Omron Sysmac Studio project distributing_station_with_timer_1.9_attempt (Sysmac Studio 1.54.0.64019, StandardProject)

# Controller new_Controller_0: NJ301-1100 version 1.14
Units and slaves: Node1 : NX-ECC201 (E001); Unit 1 : NX-PC0020 (N1); Unit 2 : NX-ID5442 (N2); Unit 3 : NX-PC0010 (N3); Unit 4 : NX-PC0020 (N4); Unit 5 : NX-OD5121 (N5); Unit 6 : NX-PC0010 (N6); Power Supply : NJ-Px3001; CPU : NJ301-1100; 0 [Unit 0] : CJ1W-AD041-V1 (J01); 1 [Unit 1] : CJ1W-DA041 (J02); 2 : CJ1W-ID211 (J03); 3 : CJ1W-OC211 (J04)
Task PrimaryTask (priority 4, period or condition 1000): Program0

VAR_GLOBAL
    Station_1B2 : BOOL;  (* Ejection Cylinder Extended; at IOBus://rack#0/slot#2/Ch1_In/Ch1_In01; published *)
    Station_1B1 : BOOL;  (* Ejection Cylinder retracted; at IOBus://rack#0/slot#2/Ch1_In/Ch1_In02; published *)
    Station_2B1 : BOOL;  (* Workpiece gripped; at IOBus://rack#0/slot#2/Ch1_In/Ch1_In03; published *)
    Station_3S1 : BOOL;  (* arm_in_magazine; at IOBus://rack#0/slot#2/Ch1_In/Ch1_In04; published *)
    Station_3S2 : BOOL;  (* arm_in_downstream; at IOBus://rack#0/slot#2/Ch1_In/Ch1_In05; published *)
    Station_B4 : BOOL;  (* Magzine empty; at IOBus://rack#0/slot#2/Ch1_In/Ch1_In06; published *)
    Panel_S1 : BOOL;  (* start_button; at IOBus://rack#0/slot#2/Ch1_In/Ch1_In08; published *)
    Panel_S2 : BOOL;  (* stop_button; at IOBus://rack#0/slot#2/Ch1_In/Ch1_In09; published *)
    Panel_S4 : BOOL;  (* reset_button; at IOBus://rack#0/slot#2/Ch1_In/Ch1_In11; published *)
    Station_1Y1 : BOOL;  (* Magzine eject; at IOBus://rack#0/slot#3/Ch1_Out/Ch1_Out00; published *)
    Station_2Y1 : BOOL;  (* Vacuum on; at IOBus://rack#0/slot#3/Ch1_Out/Ch1_Out01; published *)
    Station_2Y2 : BOOL;  (* Ejector_Pulse_On; at IOBus://rack#0/slot#3/Ch1_Out/Ch1_Out02; published *)
    Station_3Y1 : BOOL;  (* arm_2_magazine; at IOBus://rack#0/slot#3/Ch1_Out/Ch1_Out03; published *)
    Station_3Y2 : BOOL;  (* arm_2_downstream; at IOBus://rack#0/slot#3/Ch1_Out/Ch1_Out04; published *)
    Station_H1 : BOOL;  (* start light; at IOBus://rack#0/slot#3/Ch1_Out/Ch1_Out08; published *)
    Station_H2 : BOOL;  (* reset light; at IOBus://rack#0/slot#3/Ch1_Out/Ch1_Out09; published *)
    Panel_H3 : BOOL;  (* Q1 light; at IOBus://rack#0/slot#3/Ch1_Out/Ch1_Out10; published *)
    Panel_H4 : BOOL;  (* Q2 light; at IOBus://rack#0/slot#3/Ch1_Out/Ch1_Out11; published *)
    Station_1B1_in : BOOL;
END_VAR

PROGRAM Program0
VAR
    FB_Panel_1 : FB_Panel;
    run_mode : BOOL;
    stop_mode : BOOL;
    reset_mode : BOOL;
    FB_Actuator_T1_1 : FB_Actuator_T1;
    timer_t1 : TON;
    error_arm : BOOL;
    error_mode : BOOL;
    FB_Actuator_T2_1 : FB_Actuator_T2;
    Piston : RS;
    error_ejec : BOOL;
    extend_piston : BOOL;
    workpiece_ready_set : BOOL;
    flip_flop_1 : RS;
    workpiece_ready : BOOL;
    workpiece_picked_up : BOOL;
    wait_for_piston : TON;
    Workpiece_Checker_1 : Workpiece_Checker;
END_VAR
VAR_EXTERNAL
    Station_3S1 : BOOL;
    Panel_S2 : BOOL;
    Station_3Y2 : BOOL;
    Station_3S2 : BOOL;
    Panel_S1 : BOOL;
    Station_3Y1 : BOOL;
    Panel_S4 : BOOL;
    Station_H1 : BOOL;
    Station_H2 : BOOL;
    Panel_H4 : BOOL;
    Panel_H3 : BOOL;
    Station_1B2 : BOOL;
    Station_1B1 : BOOL;
    Station_1Y1 : BOOL;
    Station_2Y1 : BOOL;
END_VAR
VAR
    _e1 : F_TRIG;
END_VAR

(* Section Section0: ladder, written here as Structured Text *)

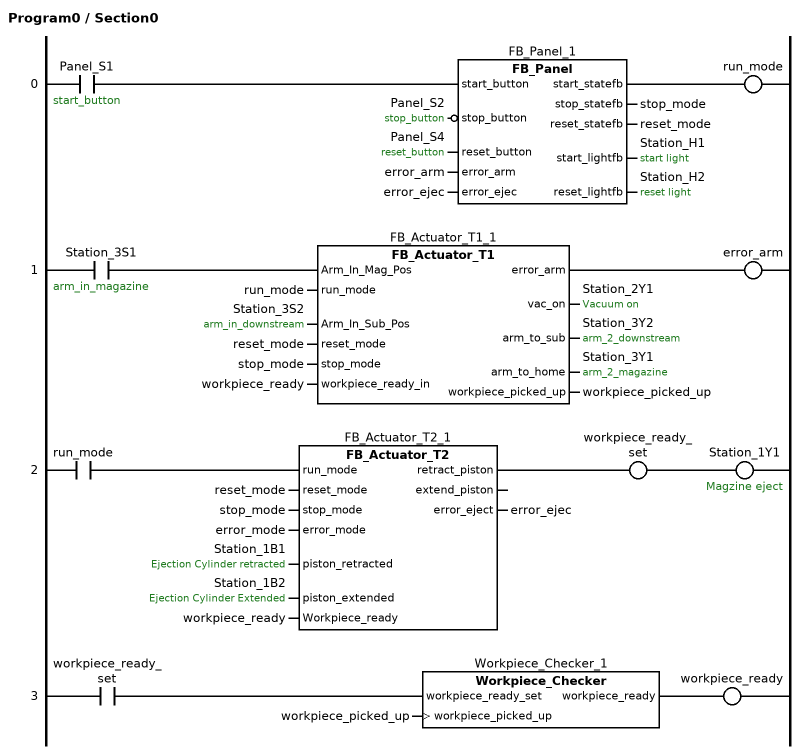
(* Rung 0 *)
FB_Panel_1(start_button := Panel_S1, stop_button := NOT Panel_S2, reset_button := Panel_S4, error_arm := error_arm, error_ejec := error_ejec, stop_statefb => stop_mode, reset_statefb => reset_mode, start_lightfb => Station_H1, reset_lightfb => Station_H2);
run_mode := FB_Panel_1.start_statefb;
(* Rung 1 *)
FB_Actuator_T1_1(Arm_In_Mag_Pos := Station_3S1, run_mode := run_mode, Arm_In_Sub_Pos := Station_3S2, reset_mode := reset_mode, stop_mode := stop_mode, workpiece_ready_in := workpiece_ready, vac_on => Station_2Y1, arm_to_sub => Station_3Y2, arm_to_home => Station_3Y1, workpiece_picked_up => workpiece_picked_up);
error_arm := FB_Actuator_T1_1.error_arm;
(* Rung 2 *)
FB_Actuator_T2_1(run_mode := run_mode, reset_mode := reset_mode, stop_mode := stop_mode, error_mode := error_mode, piston_retracted := Station_1B1, piston_extended := Station_1B2, Workpiece_ready := workpiece_ready, error_eject => error_ejec);
workpiece_ready_set := FB_Actuator_T2_1.retract_piston;
Station_1Y1 := FB_Actuator_T2_1.retract_piston;
(* Rung 3 *)
_e1(CLK := workpiece_picked_up);
Workpiece_Checker_1(workpiece_ready_set := workpiece_ready_set, workpiece_picked_up := _e1.Q);
workpiece_ready := Workpiece_Checker_1.workpiece_ready;
END_PROGRAM

FUNCTION_BLOCK FB_Panel
VAR
    flip_flop : RS;
    flip_flop2 : RS;
    flip_flop_3 : RS;
    flip_flop3 : RS;
    stop_or_error : BOOL;
    error_armfb : BOOL;
    error_q2 : BOOL;
END_VAR
VAR_OUTPUT
    start_statefb : BOOL;
    stop_statefb : BOOL;
    reset_statefb : BOOL;
END_VAR
VAR_INPUT
    start_button : BOOL := False;
    stop_button : BOOL := False;
    reset_button : BOOL := False;
END_VAR
VAR_OUTPUT
    start_lightfb : BOOL;
    reset_lightfb : BOOL;
END_VAR
VAR_INPUT
    error_arm : BOOL;
    error_ejec : BOOL;
END_VAR
VAR_EXTERNAL
    Panel_H4 : BOOL;
END_VAR
(* ladder, written here as Structured Text *)

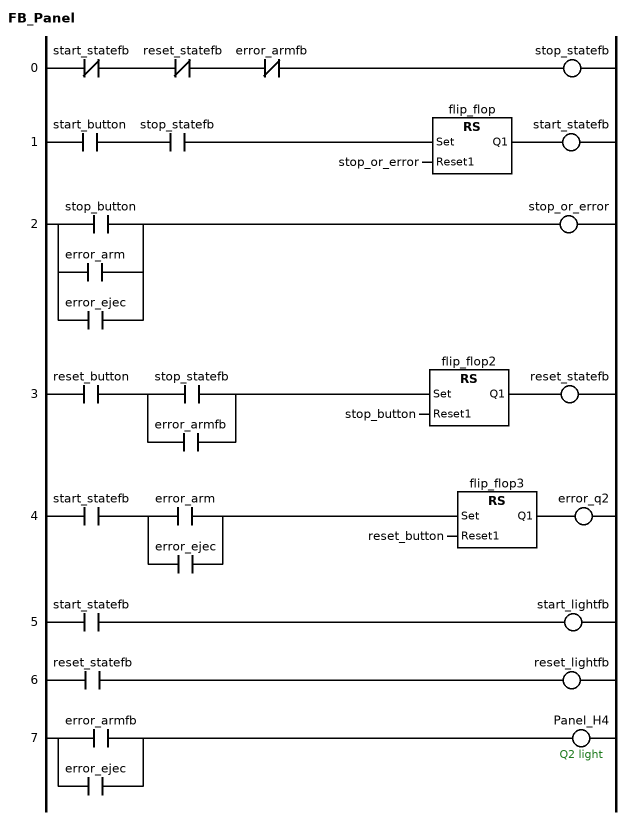
(* Rung 0 *)
stop_statefb := NOT start_statefb AND NOT reset_statefb AND NOT error_armfb;
(* Rung 1 *)
flip_flop(Set := start_button AND stop_statefb, Reset1 := stop_or_error);
start_statefb := flip_flop.Q1;
(* Rung 2 *)
stop_or_error := stop_button OR error_arm OR error_ejec;
(* Rung 3 *)
flip_flop2(Set := reset_button AND (stop_statefb OR error_armfb), Reset1 := stop_button);
reset_statefb := flip_flop2.Q1;
(* Rung 4 *)
flip_flop3(Set := start_statefb AND (error_arm OR error_ejec), Reset1 := reset_button);
error_q2 := flip_flop3.Q1;
(* Rung 5 *)
start_lightfb := start_statefb;
(* Rung 6 *)
reset_lightfb := reset_statefb;
(* Rung 7 *)
Panel_H4 := error_armfb OR error_ejec;
END_FUNCTION_BLOCK

FUNCTION_BLOCK FB_Actuator_T1
VAR
    flip_flop_1 : RS;
    flip_flop_2 : RS;
    reset_to_home : BOOL;
    timer_t1 : TON;
    flip_flop_3 : RS;
    timer_t2 : TON;
    flip_flop_4 : RS;
    error_toSub : BOOL;
    error_toHome : BOOL;
    middle_pos : BOOL;
    middle_timer : AccumulationTimer;
    flip_flop_5 : RS;
    reset_middle : BOOL;
    flip_flop6 : RS;
    move_to_middle_from_home : BOOL;
    move_to_sub : BOOL;
    move_to_home : BOOL;
    move_to_middle_from_sub : BOOL;
    unknown_pos : BOOL;
    reset_vac_arm_to_sub : BOOL;
    timer_t3 : TON;
    t : TIME;
    move_to_su : BOOL;
END_VAR
VAR_INPUT
    Arm_In_Mag_Pos : BOOL;
    run_mode : BOOL;
    Arm_In_Sub_Pos : BOOL;
    reset_mode : BOOL;
    stop_mode : BOOL;
END_VAR
VAR_OUTPUT
    error_arm : BOOL;
END_VAR
VAR_INPUT
    workpiece_ready_in : BOOL;
END_VAR
VAR_OUTPUT
    vac_on : BOOL;
    arm_to_sub : BOOL;
    arm_to_home : BOOL;
    workpiece_picked_up : BOOL;
END_VAR
VAR_EXTERNAL
    Station_3S1 : BOOL;
    Station_3Y1 : BOOL;
    Station_3S2 : BOOL;
    Station_3Y2 : BOOL;
    Station_2Y2 : BOOL;
END_VAR
(* ladder, written here as Structured Text *)

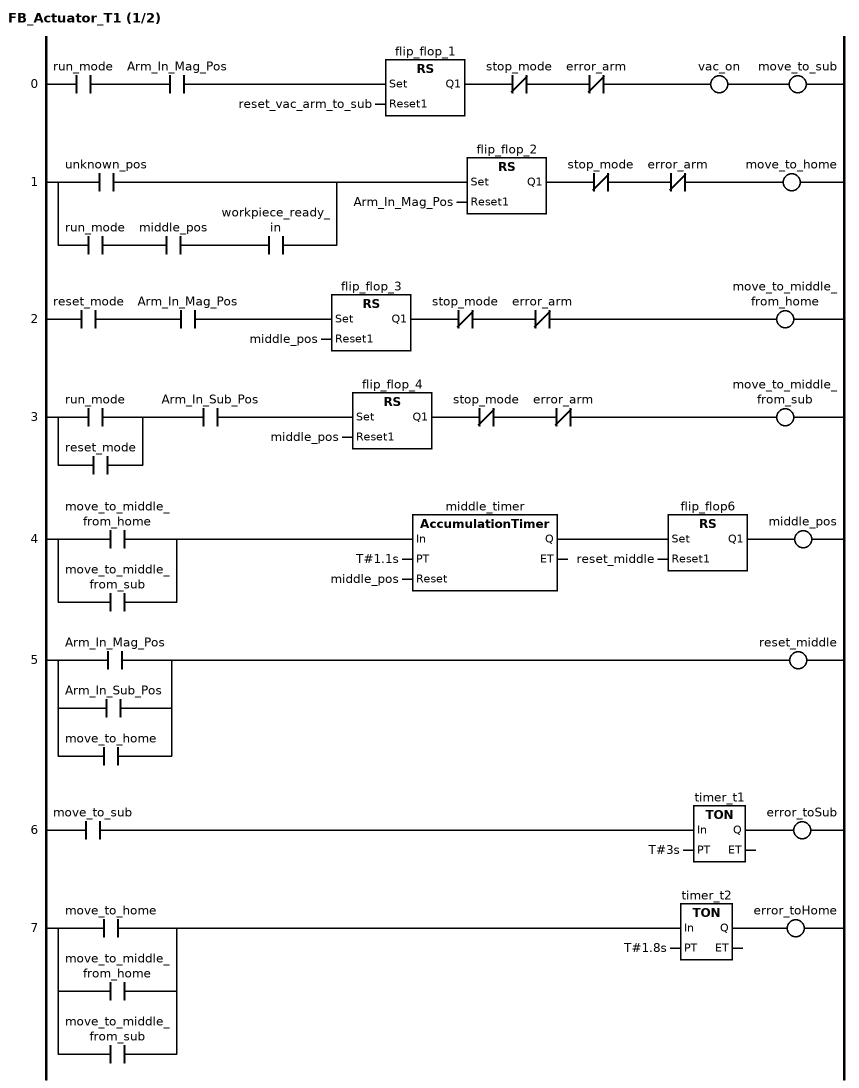
(* Rung 0 *)
flip_flop_1(Set := run_mode AND Arm_In_Mag_Pos, Reset1 := reset_vac_arm_to_sub);
vac_on := flip_flop_1.Q1 AND NOT stop_mode AND NOT error_arm;
move_to_sub := flip_flop_1.Q1 AND NOT stop_mode AND NOT error_arm;
(* Rung 1 *)
flip_flop_2(Set := unknown_pos OR (run_mode AND middle_pos AND workpiece_ready_in), Reset1 := Arm_In_Mag_Pos);
move_to_home := flip_flop_2.Q1 AND NOT stop_mode AND NOT error_arm;
(* Rung 2 *)
flip_flop_3(Set := reset_mode AND Arm_In_Mag_Pos, Reset1 := middle_pos);
move_to_middle_from_home := flip_flop_3.Q1 AND NOT stop_mode AND NOT error_arm;
(* Rung 3 *)
flip_flop_4(Set := (run_mode OR reset_mode) AND Arm_In_Sub_Pos, Reset1 := middle_pos);
move_to_middle_from_sub := flip_flop_4.Q1 AND NOT stop_mode AND NOT error_arm;
(* Rung 4 *)
middle_timer(In := move_to_middle_from_home OR move_to_middle_from_sub, PT := T#1.1s, Reset := middle_pos);
flip_flop6(Set := middle_timer.Q, Reset1 := reset_middle);
middle_pos := flip_flop6.Q1;
(* Rung 5 *)
reset_middle := Arm_In_Mag_Pos OR Arm_In_Sub_Pos OR move_to_home;
(* Rung 6 *)
timer_t1(In := move_to_sub, PT := T#3s);
error_toSub := timer_t1.Q;
(* Rung 7 *)
timer_t2(In := move_to_home OR move_to_middle_from_home OR move_to_middle_from_sub, PT := T#1.8s);
error_toHome := timer_t2.Q;

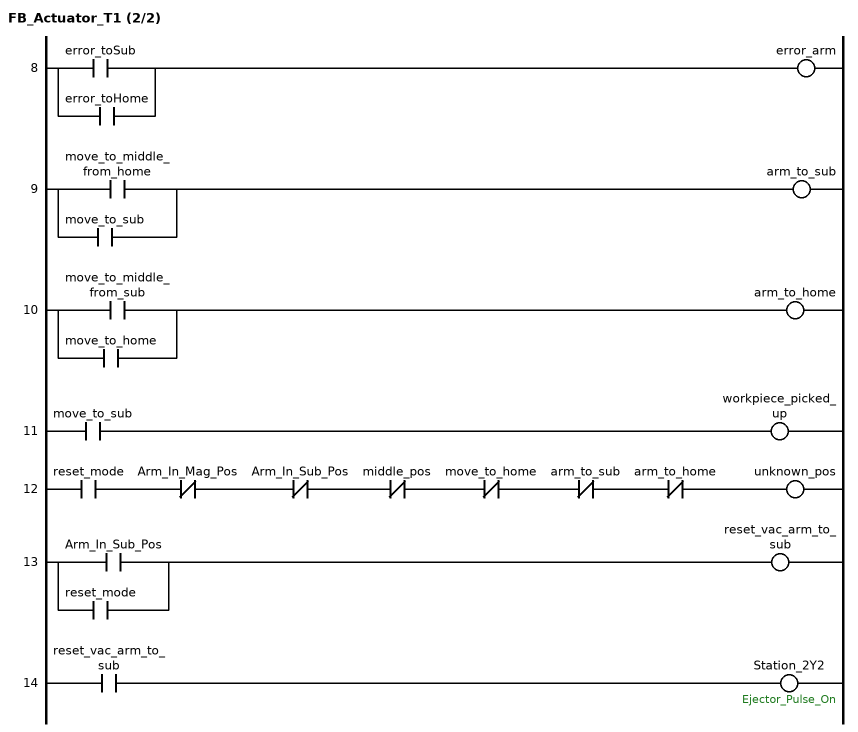
(* Rung 8 *)
error_arm := error_toSub OR error_toHome;
(* Rung 9 *)
arm_to_sub := move_to_middle_from_home OR move_to_sub;
(* Rung 10 *)
arm_to_home := move_to_middle_from_sub OR move_to_home;
(* Rung 11 *)
workpiece_picked_up := move_to_sub;
(* Rung 12 *)
unknown_pos := reset_mode AND NOT Arm_In_Mag_Pos AND NOT Arm_In_Sub_Pos AND NOT middle_pos AND NOT move_to_home AND NOT arm_to_sub AND NOT arm_to_home;
(* Rung 13 *)
reset_vac_arm_to_sub := Arm_In_Sub_Pos OR reset_mode;
(* Rung 14 *)
Station_2Y2 := reset_vac_arm_to_sub;
END_FUNCTION_BLOCK

FUNCTION_BLOCK FB_Actuator_T2
VAR
    reset_to_home : BOOL;
    retract_ff : RS;
    extend_ff : RS;
    extend_t : TON;
    retract_t : TON;
    retract_err : BOOL;
    extend_err : BOOL;
    workpiece_lifted : BOOL;
    Workpiece_ejection : RS;
END_VAR
VAR_INPUT
    run_mode : BOOL;
    reset_mode : BOOL;
    stop_mode : BOOL;
    error_mode : BOOL;
END_VAR
VAR_OUTPUT
    retract_piston : BOOL;
    extend_piston : BOOL;
END_VAR
VAR_INPUT
    piston_retracted : BOOL;
    piston_extended : BOOL;
END_VAR
VAR_OUTPUT
    error_eject : BOOL;
END_VAR
VAR_INPUT
    Workpiece_ready : BOOL;
END_VAR
VAR_EXTERNAL
    Station_B4 : BOOL;
    Station_1B1 : BOOL;
    Station_1B2 : BOOL;
    Station_2Y1 : BOOL;
END_VAR
(* ladder, written here as Structured Text *)

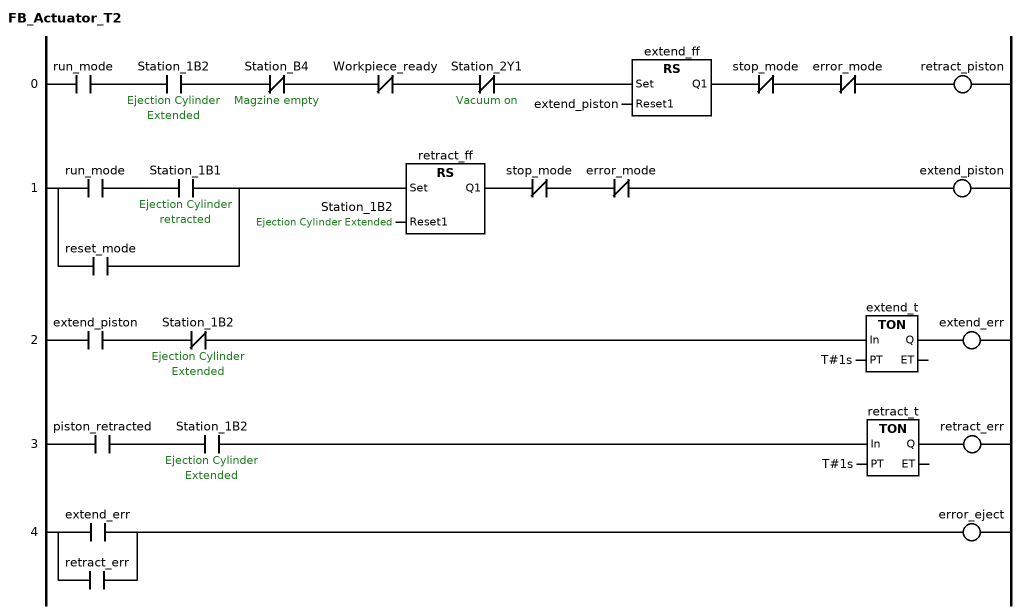
(* Rung 0 *)
extend_ff(Set := run_mode AND Station_1B2 AND NOT Station_B4 AND NOT Workpiece_ready AND NOT Station_2Y1, Reset1 := extend_piston);
retract_piston := extend_ff.Q1 AND NOT stop_mode AND NOT error_mode;
(* Rung 1 *)
retract_ff(Set := (run_mode AND Station_1B1) OR reset_mode, Reset1 := Station_1B2);
extend_piston := retract_ff.Q1 AND NOT stop_mode AND NOT error_mode;
(* Rung 2 *)
extend_t(In := extend_piston AND NOT Station_1B2, PT := T#1s);
extend_err := extend_t.Q;
(* Rung 3 *)
retract_t(In := piston_retracted AND Station_1B2, PT := T#1s);
retract_err := retract_t.Q;
(* Rung 4 *)
error_eject := extend_err OR retract_err;
END_FUNCTION_BLOCK

FUNCTION_BLOCK Workpiece_Checker
VAR
    wait_for_piston : TON;
    flip_flop_1 : RS;
END_VAR
VAR_INPUT
    workpiece_ready_set : BOOL;
    workpiece_picked_up : BOOL (* edge DownDirection *);
END_VAR
VAR_OUTPUT
    workpiece_ready : BOOL;
END_VAR
(* ladder, written here as Structured Text *)

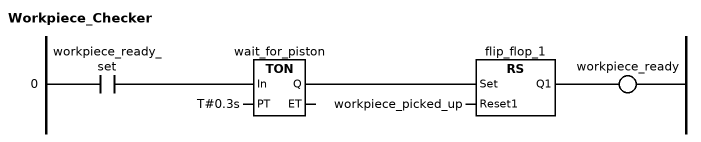
(* Rung 0 *)
wait_for_piston(In := workpiece_ready_set, PT := T#0.3s);
flip_flop_1(Set := wait_for_piston.Q, Reset1 := workpiece_picked_up);
workpiece_ready := flip_flop_1.Q1;
END_FUNCTION_BLOCK